PROGRAM PRG_PMPS
VAR
    fbArbiterIO : FB_SubSysToArbiter_IO;

END_VAR

fbArbiterIO(Arbiter := g_fbArbiter1, fbFFHWO := g_FastFaultOutput1);
g_fbArbiter1.AddRequest(nReqID := 95 , stReqBp := PMPS_GVL.cstFullBeam, sDevName := 'plc-lfe-vac');

(*FastFaultOuput*)
g_FastFaultOutput1.Execute(bAutoReset:= TRUE);
g_FastFaultOutput2.Execute(i_xVeto:=PMPS_GVL.stCurrentBeamParameters.aVetoDevices[PMPS.L_Stopper.ST1L0], bAutoReset:= TRUE);

END_PROGRAM

(* stored: Version 1.1.0.1, ProductVersion 3.1.4022.18
   POU PRG_PMPS: Id {10012da2-da02-4fd4-92c9-6bee3a2cc733}, SpecialFunc None *)
